FUNCTION_BLOCK FB_SortingModule EXTENDS FB_SubsystemRoot
VAR_INPUT
	bButtonCylMoveToWorkIn										:						BOOL;
	bButtonCylMoveToBaseIn										:						BOOL;
END_VAR
VAR_OUTPUT
	bSorted														:						BOOL;								// Part picked at sorting module
	
	bCylError													:						BOOL;
	sCylErrorMsg												:						STRING;
	
	aCylTemps													:						ARRAY [1..100] OF LREAL;
	
	bButtonCylMoveToWorkOut										:						BOOL;
	bButtonCylMoveToBaseOut										:						BOOL;
END_VAR
VAR
	// Sensor with delay functionality
	fbSensorDelay												:						FB_SignalHandlingDelay;
	
	// Function block instance for cylinder
	fbCylinder													:						FB_CylinderBase;
	fbCylinderDiag												:						FB_CylinderDiag;
	fbCylinderTemp												:						FB_CylinderTemp;
	fbCylinderTempDiag											:						FB_CylinderTempDiag;
	fbCylinderTempRec											:						FB_CylinderTempRecord;
	// Interface instance for cylinder
	itfCylinder													:						I_Cylinder;
	// Time parameters for submodules
	tTimeOutCylinder											:						TIME;								// For cylinder with position diagnosis: time in which the cylinder shcould reach work / base position
	tTimeIntervalCylinder										:						TIME;								// Time of intervals to record the temperature of cylinder
	tSensorDelay												:						TIME;								// Sensor delay
	tMoveAxisDelay												:						TIME;								// Time delay to stop running axis
	// ========================== Temperature parameters for cylinder  ======================================================================
	nTempMinCyl													:						LREAL;								// For cylinder with temperature diagnosis: minimal temperature
	nTempMaxCyl													:						LREAL;								// For cylinder with temperature diagnosis: maximal temperature
	// Manual cylinder controll
	fbButtonCylMoveToWork										:						FB_SignalHandlingIntern;			// Button to move cylinder manually to work position
	fbButtonCylMoveToBase										:						FB_SignalHandlingIntern;			// Button to move cylinder manually to base position
	// Common variables
	fbTimerAxis													:						TON;								// Timer to run axis for certain amount of time
	fbTriggerCylAtWorkPos										:						R_TRIG;								// Trigger to recognize rising edge of cylinder being at work position
	eStateAutoAxis												:						E_StateSortingAutoAxis;				// State variable for automatic / semi-auto mode for axis movement
	eStateAutoCylinder											:						E_StateSortingAutoCylinder;			// State variable for automatic / semi-auto mode for cylinder movement
END_VAR

METHOD Automatic
VAR_INPUT
END_VAR
	fbTriggerCylAtWorkPos(		CLK			:=		itfCylinder.bState_AtWorkPos);

	CASE eStateAutoAxis OF
		
		E_StateSortingAutoAxis.WaitForCylinderAtWorkPos:
			IF fbTriggerCylAtWorkPos.Q THEN
				fbTimerAxis(	IN			:=		TRUE,
								PT			:=		tMoveAxisDelay);
				
				eStateAutoAxis				:=		E_StateSortingAutoAxis.MoveAxis;
			END_IF
		
		E_StateSortingAutoAxis.MoveAxis:
			fbTimerAxis();
			IF bHaltRequest THEN
				
				eStateAutoAxis				:=		E_StateSortingAutoAxis.StopAxis;
			ELSIF fbTimerAxis.Q THEN
				fbTimerAxis(	IN			:=		FALSE);
				
				bSorted						:=		TRUE;
			
				eStateAutoAxis				:=		E_StateSortingAutoAxis.StopAxis;
			ELSE
				fbAxis.MoveFw();
			END_IF
		
		E_StateSortingAutoAxis.StopAxis:
				bSorted						:=		FALSE;
				
				IF NOT bHaltDone THEN
					Stop(	bStop			:=		TRUE);
				ELSE	
					Stop(	bStop			:=		FALSE);
					eStateAutoAxis			:=		E_StateSortingAutoAxis.WaitForCylinderAtWorkPos;
				END_IF   
	END_CASE
	
	CASE eStateAutoCylinder OF
		E_StateSortingAutoCylinder.BoxDetected:
		
			itfCylinder.MoveToBase();
			
			IF fbSensorDelay.bOutputSignal THEN
				eStateAutoCylinder			:=		E_StateSortingAutoCylinder.MoveCylToWorkPos;	
			END_IF
				
		E_StateSortingAutoCylinder.MoveCylToWorkPos:
		
			itfCylinder.MoveToWork();
			
			IF itfCylinder.bState_AtWorkPos THEN
				eStateAutoCylinder			:=		E_StateSortingAutoCylinder.MoveCylToBasePos;
			END_IF
			
		E_StateSortingAutoCylinder.MoveCylToBasePos:
			itfCylinder.MoveToBase();
			
			IF itfCylinder.bState_AtBasePos THEN
				eStateAutoCylinder			:=		E_StateSortingAutoCylinder.BoxDetected;
			END_IF	
	END_CASE
END_METHOD

PROPERTY bState_CylAtBasePos : BOOL
GET
bState_CylAtBasePos			:=		itfCylinder.bState_AtBasePos;
END_GET
END_PROPERTY

PROPERTY bState_CylAtWorkPos : BOOL
GET
bState_CylAtWorkPos			:=		itfCylinder.bState_AtWorkPos;
END_GET
END_PROPERTY

METHOD CylinderOptions
VAR_INPUT
	bCylDiag							:				BOOL;						// If TRUE cylinder has diagnostic functionality
	bCylTemp							:				BOOL;						// If TRUE cylinder has temperature functionality
	bCylRecord							:				BOOL;						// If TRUE cylinder has record functionality
END_VAR

	IF 	bCylDiag THEN
		IF bCylTemp THEN
			fbCylinderTempDiag.fTempMin				:=			nTempMinCyl;
			fbCylinderTempDiag.fTempMax				:=			nTempMaxCyl;
			bCylError								:=			fbCylinderTempDiag.bError;
			sCylErrorMsg							:=			fbCylinderTempDiag.sErrorMsg;
				itfCylinder								:=			fbCylinderTempDiag;
		ELSE
			bCylError								:=			fbCylinderDiag.bError;
			sCylErrorMsg							:=			fbCylinderDiag.sErrorMsg;
			fbCylinderDiag.nTimeOut					:=			tTimeOutCylinder;			
				itfCylinder								:=			fbCylinderDiag;
		END_IF
	ELSE
		bCylError									:=			FALSE;
		sCylErrorMsg								:=			'';
		
		IF 	bCylTemp THEN
			IF bCylRecord THEN
				fbCylinderTempRec.nTimeInterval		:=			tTimeIntervalCylinder;
				fbCylinderTempRec.bRecordStart		:=			bCompresAirEnableLocal;
				
				fbCylinderTempRec.Record();
				
				aCylTemps							:=			fbCylinderTempRec.aRecords;
				
					itfCylinder	:= fbCylinderTempRec;
			
			ELSE
					itfCylinder	:=	fbCylinderTemp;
			END_IF
		ELSE
					itfCylinder	:= fbCylinder;
		END_IF
			
	END_IF
	
	;
END_METHOD

METHOD Enable
VAR_INPUT
	bComprAirEnable					:			BOOL;			// Enable of compressed air
	bAxisEnable						:			BOOL;			// Enable of axis
	bSensorEnable					:			BOOL;			// Enable of sensor
	bManualAxisEnable				:			BOOL;			// Enable manual axis control
END_VAR

VAR
	bManualEnable: BOOL;
END_VAR

	SUPER^.Enable(	bComprAirEnable				:=	bComprAirEnable,
					bAxisEnable					:=	bAxisEnable,
					bSensorEnable				:=	bSensorEnable,
					bManualAxisEnable			:=	bManualAxisEnable);
					
	fbSensorDelay.Enable(bEnable				:=	bSensorEnable);
	
	fbButtonCylMoveToWork.Enable(bEnable		:=	bManualCylinderEnableLocal AND NOT itfCylinder.bState_AtWorkPos);					// bManualAxisEnableLocal AND bComprAirEnabledLocal	
	fbButtonCylMoveToBase.Enable(bEnable		:=	bManualCylinderEnableLocal AND NOT itfCylinder.bState_AtBasePos);					// bManualAxisEnableLocal AND bComprAirEnabledLocal
	
	fbButtonCylMoveToWork.bInputSignal			:=	NOT fbButtonCylMoveToBase.bInputSignal;
END_METHOD

METHOD InputOutput
VAR_INPUT
END_VAR

	SUPER^.InputOutput();
	
	fbSensorDelay.SetOutput();
	
	
	
	fbButtonCylMoveToWork.SetOutput();
	fbButtonCylMoveToBase.SetOutput();
	
	fbButtonCylMoveToWork.bInputSignal					:=		bButtonCylMoveToWorkIn;
	fbButtonCylMoveToBase.bInputSignal					:=		bButtonCylMoveToBaseIn;
	
	bButtonCylMoveToWorkOut								:=		fbButtonCylMoveToWork.bOutputSignal;
	bButtonCylMoveToBaseOut								:=		fbButtonCylMoveToBase.bOutputSignal;
END_METHOD

METHOD Maintenance
VAR_INPUT
END_VAR

	THIS^.Manual();
END_METHOD

METHOD Manual
VAR_INPUT
END_VAR
	
	SUPER^.Manual();
	
	IF fbButtonCylMoveToWork.bOutputSignal THEN
		itfCylinder.MoveToWork();
	ELSIF	fbButtonCylMoveToBase.bOutputSignal THEN
		itfCylinder.MoveToBase();
	END_IF
END_METHOD

PROPERTY nProp_CylTempMax : LREAL
GET
nProp_CylTempMax		:=		nTempMaxCyl;
END_GET
SET
nTempMaxCyl			:=		nProp_CylTempMax;
END_SET
END_PROPERTY

PROPERTY nProp_CylTempMin : LREAL
GET
nProp_CylTempMin		:=		nTempMinCyl;
END_GET
SET
nTempMinCyl			:=		nProp_CylTempMin;
END_SET
END_PROPERTY

METHOD Reset
VAR_INPUT
	bReset				:			BOOL;			// True if machine is in state RESETTING
END_VAR

	SUPER^.Reset(	bReset			:=			bReset);
	
	IF fbTriggerResetStart.Q THEN
	
	fbTimerAxis(	IN				:=			FALSE);			
	
	itfCylinder.Reset();
	
	END_IF
END_METHOD

METHOD ResetState
VAR_INPUT
END_VAR
// =========================================================
	eStateAutoAxis					:=			E_StateSortingAutoAxis.WaitForCylinderAtWorkPos;
	eStateAutoCylinder				:=			E_StateSortingAutoCylinder.BoxDetected;
// =========================================================
END_METHOD

METHOD Semiautomatic
VAR_INPUT
END_VAR
	
	THIS^.Automatic();
END_METHOD

METHOD Starting
VAR_INPUT
	bStarting					:				BOOL;			// True if machine is in state STARTING
END_VAR

	SUPER^.Starting(	bStarting			:=			bStarting);
	
	fbSensorDelay.tDelay					:=			tSensorDelay;
END_METHOD

PROPERTY tProp_AxisMoving : TIME
GET
tProp_AxisMoving		:=		tMoveAxisDelay;
END_GET
SET
tMoveAxisDelay			:=		tProp_AxisMoving;
END_SET
END_PROPERTY

PROPERTY tProp_CylRecInterval : TIME
GET
tProp_CylRecInterval		:=			tTimeIntervalCylinder;
END_GET
SET
tTimeIntervalCylinder			:=			tProp_CylRecInterval;
END_SET
END_PROPERTY

PROPERTY tProp_CylTimeOut : TIME
GET
tProp_CylTimeOut			:=			tTimeOutCylinder;
END_GET
SET
tTimeOutCylinder		:=			tProp_CylTimeOut;
END_SET
END_PROPERTY

PROPERTY tProp_SensorDelay : TIME
GET
tProp_SensorDelay			:=			fbSensorDelay;
END_GET
SET
fbSensorDelay			:=			tProp_SensorDelay;
END_SET
END_PROPERTY

END_FUNCTION_BLOCK

(* stored: Version 1.1.0.1, ProductVersion 3.1.4024.15
   POU FB_SortingModule: Id {78f5a34d-589b-4d90-87e2-81c612568f87}, SpecialFunc None
   Method Automatic: Id {047bbba3-2625-45bf-ac3b-0a710f32d1ef}
   Property bState_CylAtBasePos: Id {b753a032-f87a-4904-afe1-28dcdab709dc}
   Get Get: Id {634187d1-99f7-49a2-abe8-b8ba9aa7be04}
   Property bState_CylAtWorkPos: Id {92ec6e92-9efc-4b11-964d-502576d997f2}
   Get Get: Id {7d42194f-d639-443c-8958-075057a69b3a}
   Method CylinderOptions: Id {b347b23e-806d-431e-8710-b8d7a9ff9ab5}
   Method Enable: Id {1639f444-8504-4240-9b3f-3b669453f42b}
   Method InputOutput: Id {0217b8cf-d36c-4c0f-b2a1-28b45245a175}
   Method Maintenance: Id {770913ac-2b66-445d-b7d1-73a1f828a233}
   Method Manual: Id {d2cefb4b-0c9f-4969-bd55-5fe4f896fcf2}
   Property nProp_CylTempMax: Id {48992803-0bd1-4afc-a370-69cd8bd0bdc7}
   Get Get: Id {96f08428-9c4d-407f-b5ba-2c5ac5d0ed57}
   Set Set: Id {15cda981-a350-418b-a615-088e59540c7b}
   Property nProp_CylTempMin: Id {baf62ffc-b88e-4ea6-af5b-ecacc8eca619}
   Get Get: Id {cc8bd3da-56b2-4d54-9440-4621c7be64d5}
   Set Set: Id {a64c9960-6a75-44e8-8562-2ddb891289d2}
   Method Reset: Id {bcef8413-fcb8-493a-a14e-8cc16a459990}
   Method ResetState: Id {1b1f2c60-74b1-49ba-8057-12522e8a424b}
   Method Semiautomatic: Id {508b12d8-8b5e-4908-aaf1-ed38e7c55eae}
   Method Starting: Id {486ca9e3-8b83-46fc-8ffd-7ee02073dc69}
   Property tProp_AxisMoving: Id {f6e230a7-8475-4329-8af5-327c8e9c17da}
   Get Get: Id {be6c9c1f-deb7-4911-b34b-11146febe38b}
   Set Set: Id {c3f55750-229d-4bf1-8ca2-6b895eee23a1}
   Property tProp_CylRecInterval: Id {cb8918e5-f9cc-4c63-8fa7-59c624786535}
   Get Get: Id {1eddf5d7-f0fc-4299-85bf-901d9874def3}
   Set Set: Id {941b3763-780f-444b-a8cf-ae71672b5785}
   Property tProp_CylTimeOut: Id {474eedd5-19a7-4f7b-9714-588a2833dc6e}
   Get Get: Id {5bf1002b-0d3c-4641-9f40-b1b40ff2737b}
   Set Set: Id {ec0d092e-bfc2-4626-b0f4-6c3db17a487c}
   Property tProp_SensorDelay: Id {d6d6e6e7-8e21-4eff-8657-b1688c617be5}
   Get Get: Id {fff513c7-0a17-4baa-9bcf-603b917b221d}
   Set Set: Id {d20fdeec-4c9a-48f9-bb4b-e58602584d3d} *)
